// TwinCAT 3 PLC project PLC1
// ProgramVersion: 3.1.4022.2
// libraries:
//   Tc2_DALI, * (Beckhoff Automation GmbH)
//   Tc2_EnOcean, * (Beckhoff Automation GmbH)
//   Tc2_IoFunctions, * (Beckhoff Automation GmbH)
//   Tc2_ModbusRTU, * (Beckhoff Automation GmbH)
//   Tc2_ModbusSrv, * (Beckhoff Automation GmbH)
//   Tc2_Standard, * (Beckhoff Automation GmbH)
//   Tc2_System, * (Beckhoff Automation GmbH)
//   Tc3_Module, * (Beckhoff Automation GmbH)
//   Tc3_PLCopen_OpcUa, * (Beckhoff Automation GmbH)
//   VisuSymbols,3.5.10.0,System
// project tree:
//   / DaliComm.TcTTO, GlobalTextList.TcGTLO, IoConversionTask.TcTTO, ModbusComm.TcTTO, PlcTask.TcTTO, Visualization Manager.TcVMO (not stored)
//   DUTs/ ATV212.TcDUT, ATV212Control.TcDUT, ATV212RegAddress.TcDUT, EL3433Index.TcDUT, EL3433Measurement.TcDUT, ErrorCode.TcDUT, Fan.TcDUT, FireIgnitor.TcDUT, GrundfosMagna3.TcDUT, GrundfosRegAddress.TcDUT, stEL3433_In.TcDUT, SupplyCondition.TcDUT
//   GVLs/ ConstList.TcGVL, GVL.TcGVL, HWVar.TcGVL, Scale.TcGVL
//   POUs/BurningProcess/ BurningProcess.TcPOU, FB_OnOffTimer.TcPOU (not stored), FeederSpeedControl.TcPOU
//   POUs/CommunicationPrograms/ BackgroundComm.TcPOU, DaliCommunication.TcPOU, EL3433SyncData.TcPOU, IOConversion.TcPOU
//   POUs/EnergyFlow/ CoolingFan.TcPOU, WaterFlowControl.TcPOU
//   POUs/Lights/ EnOcean_Dali.TcPOU
//   POUs/ MAIN.TcPOU, ModbusCommunication.TcPOU
// real-time tasks:
//   TASK PlcTask: cycle T#5ms, priority 20, ADS port 350
//   TASK ModbusComm: cycle T#5ms, priority 21, ADS port 351
//   TASK IoConversionTask: cycle T#1ms, priority 10, ADS port 352
//   TASK DaliComm: cycle T#1ms, priority 15, ADS port 353
// I/O:
//   DEVICE Device 1 (EtherCAT), AmsNetId 5.42.255.222.2.1
//     Term 1 (EK1200) [EK1200-5000 EtherCAT Power supply (2A E-Bus)]
//       Term 2 (EL1008) [EL1008 8Ch. Dig. Input 24V, 3ms]
//       Term 3 (EL6021) [EL6021 Interface (RS422/485)]
//       Term 4 (EK1122) [EK1122 2 port EtherCAT junction]
//         Term 5 (EK1914) [EK1914, 2 Ch. Safety Input/Output 24V,  TwinSAFE]
//           modules: Module 1 (FSOE), Module 2 (DIO)
//           Term 6 (EL2809) [EL2809 16Ch. Dig. Output 24V, 0.5A]
//           Term 7 (EL3214) [EL3214 4Ch. Ana. Input PT100 (RTD)]
//           Term 24 (EL3204) [EL3204 4Ch. Ana. Input PT100 (RTD)]
//           Term 16 (EL9011) [EL9011 End Terminal]
//         Term 8 (EK1100) [EK1100 EtherCAT Coupler (2A E-Bus)]
//           Term 9 (EL6021) [EL6021 Interface (RS422/485)]
//           Term 10 (EL2008) [EL2008 8Ch. Dig. Output 24V, 0.5A]
//           Term 11 (EL4022) [EL4022 2Ch. Ana. Output 4-20mA, 12bit]
//           Box 12 (BK1250)
//       Term 13 (EL3433) [EL3433 3Ch. Power Measuring]
//       Term 14 (EL3433) [EL3433 3Ch. Power Measuring]
//       Box 15 (BK1250)
// variable links:
//   PLC1/PLC1 Instance <-> Device 1 (EtherCAT)/Term 1 (EK1200)/Box 15 (BK1250)
//     DaliComm Inputs/HWVar.stKL6811_in/nData <-> Term 8 (KL6811)/Channel 1/Data In
//     DaliComm Inputs/HWVar.stKL6811_in/nStatus <-> Term 8 (KL6811)/Channel 1/State
//     DaliComm Outputs/HWVar.stKL6811_out/nCtrl <-> Term 8 (KL6811)/Channel 1/Ctrl
//     DaliComm Outputs/HWVar.stKL6811_out/nData <-> Term 8 (KL6811)/Channel 1/Data Out
//     PlcTask Inputs/HWVar.st6581_in @bit 8 <-> Term 7 (KL6581)/Channel 1/Input CNODE
//     PlcTask Inputs/HWVar.st6581_in @bit {24..48 step 8} <-> Term 7 (KL6581)/Channel 1/Input DB{0..3}  (4 links)
//     PlcTask Inputs/HWVar.st6581_in @bit {56..80 step 8} <-> Term 7 (KL6581)/Channel 1/Input ID{0..3}  (4 links)
//     PlcTask Inputs/HWVar.st6581_in @bit 16 <-> Term 7 (KL6581)/Channel 1/Input ORG
//     PlcTask Inputs/HWVar.st6581_in @bit 88 <-> Term 7 (KL6581)/Channel 1/Input STATUS
//     PlcTask Inputs/HWVar.st6581_in <-> Term 7 (KL6581)/Channel 1/Status
//     PlcTask Outputs/HWVar.st6581_out <-> Term 7 (KL6581)/Channel 1/Control
//     PlcTask Outputs/HWVar.st6581_out @bit 8 <-> Term 7 (KL6581)/Channel 1/Output CNODE
//     PlcTask Outputs/HWVar.st6581_out @bit {24..48 step 8} <-> Term 7 (KL6581)/Channel 1/Output DB{0..3}  (4 links)
//     PlcTask Outputs/HWVar.st6581_out @bit {56..80 step 8} <-> Term 7 (KL6581)/Channel 1/Output ID{0..3}  (4 links)
//     PlcTask Outputs/HWVar.st6581_out @bit 16 <-> Term 7 (KL6581)/Channel 1/Output ORG
//     PlcTask Outputs/HWVar.st6581_out @bit 88 <-> Term 7 (KL6581)/Channel 1/Output STATUS
//   PLC1/PLC1 Instance <-> Device 1 (EtherCAT)/Term 1 (EK1200)/Term 13 (EL3433)
//     IoConversionTask Inputs/HWVar.EL3433_Grid[1]/dCurrent <-> PM Inputs Channel 1/Current
//     IoConversionTask Inputs/HWVar.EL3433_Grid[2]/dCurrent <-> PM Inputs Channel 2/Current
//     IoConversionTask Inputs/HWVar.EL3433_Grid[3]/dCurrent <-> PM Inputs Channel 3/Current
//     IoConversionTask Inputs/HWVar.EL3433_Grid[1]/dIndex <-> PM Inputs Channel 1/Index
//     IoConversionTask Inputs/HWVar.EL3433_Grid[2]/dIndex <-> PM Inputs Channel 2/Index
//     IoConversionTask Inputs/HWVar.EL3433_Grid[3]/dIndex <-> PM Inputs Channel 3/Index
//     IoConversionTask Inputs/HWVar.EL3433_Grid[1]/dPower <-> PM Inputs Channel 1/Active power
//     IoConversionTask Inputs/HWVar.EL3433_Grid[2]/dPower <-> PM Inputs Channel 2/Active power
//     IoConversionTask Inputs/HWVar.EL3433_Grid[3]/dPower <-> PM Inputs Channel 3/Active power
//     IoConversionTask Inputs/HWVar.EL3433_Grid[1]/dVariant <-> PM Inputs Channel 1/Variant value
//     IoConversionTask Inputs/HWVar.EL3433_Grid[2]/dVariant <-> PM Inputs Channel 2/Variant value
//     IoConversionTask Inputs/HWVar.EL3433_Grid[3]/dVariant <-> PM Inputs Channel 3/Variant value
//     IoConversionTask Inputs/HWVar.EL3433_Grid[1]/dVoltage <-> PM Inputs Channel 1/Voltage
//     IoConversionTask Inputs/HWVar.EL3433_Grid[2]/dVoltage <-> PM Inputs Channel 2/Voltage
//     IoConversionTask Inputs/HWVar.EL3433_Grid[3]/dVoltage <-> PM Inputs Channel 3/Voltage
//     IoConversionTask Outputs/HWVar.EL3433_GridIndex[1] <-> PM Outputs Channel 1/Index
//     IoConversionTask Outputs/HWVar.EL3433_GridIndex[2] <-> PM Outputs Channel 2/Index
//     IoConversionTask Outputs/HWVar.EL3433_GridIndex[3] <-> PM Outputs Channel 3/Index
//   PLC1/PLC1 Instance <-> Device 1 (EtherCAT)/Term 1 (EK1200)/Term 14 (EL3433)
//     IoConversionTask Inputs/HWVar.EL3433_Solar/dCurrent <-> PM Inputs Channel 1/Current
//     IoConversionTask Inputs/HWVar.EL3433_Solar/dIndex <-> PM Inputs Channel 1/Index
//     IoConversionTask Inputs/HWVar.EL3433_Solar/dPower <-> PM Inputs Channel 1/Active power
//     IoConversionTask Inputs/HWVar.EL3433_Solar/dVariant <-> PM Inputs Channel 1/Variant value
//     IoConversionTask Inputs/HWVar.EL3433_Solar/dVoltage <-> PM Inputs Channel 1/Voltage
//     IoConversionTask Outputs/HWVar.EL3433_SolarIndex <-> PM Outputs Channel 1/Index
//   PLC1/PLC1 Instance <-> Device 1 (EtherCAT)/Term 1 (EK1200)/Term 3 (EL6021)
//     PlcTask Inputs/HWVar.ModbusMaster1.InData @bit {16..184 step 8} <-> COM TxPDO-Map Inputs/Data In {0..21}  (22 links)
//     PlcTask Inputs/HWVar.ModbusMaster1.InData <-> COM TxPDO-Map Inputs/Status
//     PlcTask Outputs/HWVar.ModbusMaster1.OutData <-> COM RxPDO-Map Outputs/Ctrl
//     PlcTask Outputs/HWVar.ModbusMaster1.OutData @bit {16..184 step 8} <-> COM RxPDO-Map Outputs/Data Out {0..21}  (22 links)
//   PLC1/PLC1 Instance <-> Device 1 (EtherCAT)/Term 1 (EK1200)/Term 4 (EK1122)/Term 5 (EK1914)/Term 24 (EL3204)
//     IoConversionTask Inputs/HWVar.iAI2_VK[{1..4}] <-> RTD Inputs Channel {1..4}/Value  (4 links)
//   PLC1/PLC1 Instance <-> Device 1 (EtherCAT)/Term 1 (EK1200)/Term 4 (EK1122)/Term 5 (EK1914)/Term 6 (EL2809)
//     PlcTask Outputs/GVL.bFanPower <-> Channel 12/Output
//     PlcTask Outputs/GVL.bHV[{2..11}] <-> Channel {2..11}/Output  (10 links)
//     PlcTask Outputs/GVL.bHV[1] <-> Channel 1/GVL.bHV[1]
//   PLC1/PLC1 Instance <-> Device 1 (EtherCAT)/Term 1 (EK1200)/Term 4 (EK1122)/Term 5 (EK1914)/Term 7 (EL3214)
//     IoConversionTask Inputs/HWVar.iAI1_VK[{1..4}] <-> RTD Inputs Channel {1..4}/HWVar.iAI1_VK[{1..4}]  (4 links)
//   PLC1/PLC1 Instance <-> Device 1 (EtherCAT)/Term 1 (EK1200)/Term 4 (EK1122)/Term 8 (EK1100)/Box 12 (BK1250)
//     IoConversionTask Inputs/HWVar.iAI1_JK[{1..4}] <-> Term 5 (KL3204)/Channel {1..4}/Data In  (4 links)
//     IoConversionTask Inputs/HWVar.iKL3064[{1..4}] <-> Term 17 (KL3064)/Channel {1..4}/HWVar.iKL3064[{1..4}]  (4 links)
//     IoConversionTask Inputs/HWVar.stKL2761_in/iDataIn <-> Term 15 (KL2761)/Channel 1/Data In
//     IoConversionTask Inputs/HWVar.stKL2761_in/iState <-> Term 15 (KL2761)/Channel 1/State
//     IoConversionTask Inputs/HWVar.stKL3208_in/iDataIn <-> Term 3 (KL3208-0010-4)/Channel 1/Data In
//     IoConversionTask Inputs/HWVar.stKL3208_in/iState <-> Term 3 (KL3208-0010-4)/Channel 1/State
//     IoConversionTask Outputs/HWVar.stKL2761_out/iCtrl <-> Term 15 (KL2761)/Channel 1/Ctrl
//     IoConversionTask Outputs/HWVar.stKL2761_out/iDataOut <-> Term 15 (KL2761)/Channel 1/Data Out
//     ModbusComm Outputs/HWVar.stKL3204_out/iCtrl <-> Term 5 (KL3204)/Channel 4/Ctrl
//     ModbusComm Outputs/HWVar.stKL3204_out/iDataOut <-> Term 5 (KL3204)/Channel 4/Data Out
//     PlcTask Outputs/HWVar.stKL3208_out/iCtrl <-> Term 3 (KL3208-0010-4)/Channel 1/Ctrl
//     PlcTask Outputs/HWVar.stKL3208_out/iDataOut <-> Term 3 (KL3208-0010-4)/Channel 1/Data Out
//   PLC1/PLC1 Instance <-> Device 1 (EtherCAT)/Term 1 (EK1200)/Term 4 (EK1122)/Term 8 (EK1100)/Term 10 (EL2008)
//     PlcTask Outputs/GVL.stFI1/bBlower <-> Channel 5/Output
//     PlcTask Outputs/GVL.stFI1/bHeating <-> Channel 3/Output
//   PLC1/PLC1 Instance <-> Device 1 (EtherCAT)/Term 1 (EK1200)/Term 4 (EK1122)/Term 8 (EK1100)/Term 9 (EL6021)
//     PlcTask Inputs/HWVar.ModbusMaster.InData/D <-> COM TxPDO-Map Inputs/Data In 0
//     PlcTask Inputs/HWVar.ModbusMaster.InData/D @bit {8..168 step 8} <-> COM TxPDO-Map Inputs/Data In {1..21}  (21 links)
//     PlcTask Inputs/HWVar.ModbusMaster.InData/Status <-> COM TxPDO-Map Inputs/Status
//     PlcTask Outputs/HWVar.ModbusMaster.OutData/Ctrl <-> COM RxPDO-Map Outputs/Ctrl
//     PlcTask Outputs/HWVar.ModbusMaster.OutData/D <-> COM RxPDO-Map Outputs/Data Out 0
//     PlcTask Outputs/HWVar.ModbusMaster.OutData/D @bit {8..168 step 8} <-> COM RxPDO-Map Outputs/Data Out {1..21}  (21 links)

CONFIGURATION PLC1
    RESOURCE PLC ON TwinCAT3
        TASK DaliComm(INTERVAL := T#1ms, PRIORITY := 15);
        TASK IoConversionTask(INTERVAL := T#1ms, PRIORITY := 10);
        TASK ModbusComm(INTERVAL := T#5ms, PRIORITY := 21);
        TASK PlcTask(INTERVAL := T#5ms, PRIORITY := 20);
        PROGRAM DaliCommunication WITH DaliComm : DaliCommunication;
        PROGRAM IOConversion WITH IoConversionTask : IOConversion;
        PROGRAM BackgroundComm WITH ModbusComm : BackgroundComm;
        PROGRAM MAIN WITH PlcTask : MAIN;
    END_RESOURCE
END_CONFIGURATION

// ---- DUTs/ATV212.TcDUT
{attribute 'pack_mode' := '1'}
TYPE ATV212 :
STRUCT
	fMotorSpeed				: REAL;
	fOutputFrequency		: REAL;
	fOutputCurrent			: REAL;
	fOutputVoltage			: REAL;
END_STRUCT
END_TYPE

// ---- DUTs/ATV212Control.TcDUT
{attribute 'pack_mode' := '1'}
TYPE ATV212Control :
STRUCT
	bStart		: BOOL;
	bForward	: BOOL;
	fFrequency	: REAL;
	bManual		: BOOL;
	tTimeOn		: TIME;
	tTimeOff	: TIME;
END_STRUCT
END_TYPE

// ---- DUTs/ATV212RegAddress.TcDUT
{attribute 'qualified_only'}
TYPE ATV212RegAddress :
(
               listStart                        := 16#1874,
               MotorSpeed                       := 16#1875,
               Frequency                       	:= 16#1876,
               Current                        	:= 16#1877,
               Voltage                        	:= 16#1878,
               
               (*
               OutputFrequencyAtLastTrip		:= 16#FE00, // Hz Value before trip
               FrequencyReferenceBeforeRamp     := 16#FE02, // Hz Value before trip (before PI and speed ramp)
               FrequencyReferenceAfterRamp      := 16#FE15, // Hz Value before trip (after PI AND speed ramp)
               EstimatedSpeed                   := 16#FE16, // Hz Value before trip
               PIDFeedbackValue                 := 16#FE22, // Hz Value before trip
               
               
               
               Torque                           := 16#FE18,
               TorqueCurrent                    := 16#FE20,  //Value before trip
               ExcitingCurrent                  := 16#FE21,  //Value before trip*)
			   listEnd                          := 16#1879
) WORD := listStart;
END_TYPE

// ---- DUTs/EL3433Index.TcDUT
{attribute 'qualified_only'}
TYPE EL3433Index :
(	
	listStart := 3,
	ApparentPower :=3,
	Q,
	Energy,
	PF,
	Frequency,
	EnergyNegative,
	PhaseAngle,
	P1,
	S1,
	Q1,
	EnergyPositive,
	EnergyPositiveSaved,
	EnergySaved,
	EnergyNegativeSaved,
	FrequencyAvgRes,
	FrequencyHiRes,
	HeldFrequency,
	HeldFrequencyAvgRes,
	HeldFrequencyHiRes,
	listEnd := HeldFrequencyHiRes
);
END_TYPE

// ---- DUTs/EL3433Measurement.TcDUT
{attribute 'pack_mode' := '1'}
TYPE EL3433Measurement :
STRUCT
	fCurrent		: REAL;
	fVoltage		: REAL;
	fP		: REAL;
	fS		: REAL;
	fQ		: REAL;
	fEnergy		: REAL;
	fPF		: REAL;
	fFrequency		: REAL;
	fEnergyNegative		: REAL;
	fPhaseAngle		: REAL;
	fP1		: REAL;
	fS1		: REAL;
	fQ1		: REAL;
	fEnergyPositive		: REAL;
	fEnergyPositiveSaved		: REAL;
	fEnergySaved		: REAL;
	fEnergyNegativeSaved		: REAL;
	fFrequencyAvgRes		: REAL;
	fFrequencyHiRes		: REAL;
	fHeldFrequency		: REAL;
	fHeldFrequencyAvgRes		: REAL;
	fHeldFrequencyHiRes		: REAL;
END_STRUCT
END_TYPE

// ---- DUTs/ErrorCode.TcDUT
{attribute 'qualified_only'}
TYPE ErrorCode :
(
	SUCCESS := 0,
	
	// Preparation Error 
	PREPARATION_DONE := 1000,
	PREPARATION_WATER_HIGH_TEMP,
	PREPARATION_FLAME,
	PREPARATION_PUMP_NOT_CONNECTED,
	
	// Ignition Error
	IGNITION_DONE := 2000,
	IGNITION_FLAME,
	
	// Burning Error
	BURNING_DONE := 3000,
	BURNING_EMERGENCY_TEMPERATURE,
	
	// Stop Error
	STOP_ERROR	:= 4000
) UINT;
END_TYPE

// ---- DUTs/Fan.TcDUT
{attribute 'pack_mode' := '1'}
TYPE Fan :
STRUCT
	nSpeed 	: INT; // control primary fan speed 0-100%
	nTemp	: INT; // prim fan's terminal temp in Celcius
	fFE		: REAL;
END_STRUCT
END_TYPE

// ---- DUTs/FireIgnitor.TcDUT
{attribute 'pack_mode' := '1'}
TYPE FireIgnitor :
STRUCT
	bHeating				: BOOL;
	bBlower					: BOOL;
END_STRUCT
END_TYPE

// ---- DUTs/GrundfosMagna3.TcDUT
{attribute 'pack_mode' := '1'}
TYPE GrundfosMagna3 :
STRUCT
	fHead                       : REAL; 
	fVolumeFlow                 : REAL;
	fRelativePerformance        : REAL;
	fSpeed                      : REAL;
	fFrequency                  : REAL;
	fDigitalInput               : REAL;
	fDigitalOutput              : REAL;
	fActualSetpoint             : REAL;
	fMotorCurrent               : REAL;
	fDCLinkVoltage              : REAL;
	fMotorVoltage			    : REAL;
	fPower                      : REAL;
	fRemoteFlow                 : REAL;
	fInletPressure              : REAL;
    fRemotePressure             : REAL;
	fLevel                      : REAL;
	fPowerElectronicTemp        : REAL;
	fMotorTemp                  : REAL;
	fRemoteTemp                 : REAL;
	fElectronicTemp             : REAL;
	fPumpLiquidTemp             : REAL;
	fBearingTempDE			    : REAL;
	fBearingTempNDE             : REAL;
    fAuxSensorInput             : REAL;
    fSpecificEnergyConsumption  : REAL;
    fOperationTime              : REAL;         
    fTotalPoweredTime           : REAL;
    fTorque                     : REAL;
    fEnergy                     : REAL;
    fNumberOfStarts             : REAL;
    fReserved1                  : REAL;
    fRemoteTemp2                : REAL;
    fUserSetpoint               : REAL;
    fDiffPressure               : REAL;
    fOutletPressure             : REAL;
    fRemotePressure2            : REAL;
    fLoadPercent                : REAL;
    fPumpUnixRtc                : REAL;
    fMaxFlowLimit               : REAL;
    fRemoteDiffTemp             : REAL;
    fInletDiffPressure          : REAL;
    fOutletDiffPressure         : REAL;
    fRemoteDiffPressure         : REAL;
    fStorageTankLevel           : REAL;
    fAmbientTemp                : REAL;
    fHeatEnergyLifetime         : REAL;
    fHeatPower                  : REAL;
    fHeatDiffTemp               : REAL;
    fVolume                     : REAL;
    fHeatEnergyCounter2         : REAL;
    fVolume2                    : REAL;
END_STRUCT
END_TYPE

// ---- DUTs/GrundfosRegAddress.TcDUT
{attribute 'qualified_only'}
TYPE GrundfosRegAddress :
(
	listStart				   := 299,
	Head                       := 300, 
	VolumeFlow                 ,
	RelativePerformance        ,
	Speed                      ,
	Frequency                  ,
	DigitalInput               ,
	DigitalOutput              ,
	ActualSetpoint             ,
	MotorCurrent               ,
	DCLinkVoltage              ,
	MotorVoltage			   ,
	Power                      ,
	RemoteFlow                 := 313,
	InletPressure              ,
    RemotePressure             ,
	Level                      ,
	PowerElectronicTemp        ,
	MotorTemp                  ,
	RemoteTemp                 ,
	ElectronicTemp             ,
	PumpLiquidTemp             ,
	BearingTempDE			   ,
	BearingTempNDE             ,
    AuxSensorInput             ,
    SpecificEnergyConsumption  ,
    OperationTime              ,         
    TotalPoweredTime           := 328,
    Torque                     := 330,
    Energy                     ,
    NumberOfStarts             := 333,
    Reserved1                  := 335,
    RemoteTemp2                ,
    UserSetpoint               ,
    DiffPressure               ,
    OutletPressure             ,
    RemotePressure2            ,
    LoadPercent                ,
    PumpUnixRtc                ,
    MaxFlowLimit               := 344,
    RemoteDiffTemp             ,
    InletDiffPressure          ,
    OutletDiffPressure         ,
    RemoteDiffPressure         ,
    StorageTankLevel           ,
    AmbientTemp                ,
    HeatEnergyLifetime         ,
    HeatPower                  := 353,
    HeatDiffTemp               := 355,
    Volume                     ,
    HeatEnergyCounter2         := 358,
    Volume2                    := 360,
	listEnd					   := 361
) WORD := listStart;
END_TYPE

// ---- DUTs/stEL3433_In.TcDUT
{attribute 'pack_mode' := '1'}
TYPE stEL3433_In :
STRUCT
	dCurrent 	:	DINT;
	dVoltage 	:	DINT;
	dPower		:	DINT;
	dIndex 		:	USINT;
	dVariant	:	DINT;
END_STRUCT
END_TYPE

// ---- DUTs/SupplyCondition.TcDUT
{attribute 'pack_mode' := '1'}
TYPE SupplyCondition :
STRUCT
	fNeutralConductorCurrent				:REAL;
	fEnergySum				:REAL;
	fFrequency				:REAL;
	fNegativeEnergySum				:REAL;
	fPSum				:REAL;
	fSSum				:REAL;
	fQSum				:REAL;
	fFundamentalP				:REAL;
	fFundamentalS				:REAL;
	fFundamentalQ				:REAL;
	fEnergyPositive				:REAL;
	fEnergyPositiveSaved				:REAL;
	fEnergyNegative				:REAL;
	fEnergyNegativeSaved				:REAL;
	fFrequencyAvgRes				:REAL;
	fFrequencyHiRes				:REAL;
	fHeldFrequency				:REAL;
	fHeldFrequencyAvgRes				:REAL;
	fHeldFrequencyHiRes				:REAL;
	fADCTemperature				:REAL;

END_STRUCT
END_TYPE

// ---- GVLs/ConstList.TcGVL
VAR_GLOBAL
	aEL3433IndicesScale	: ARRAY[EL3433Index.listStart..EL3433Index.listEnd]	OF REAL := [
		0.01,
		0.01,
		0.001,
		0.001,
		0.1,
		0.001,
		0.01,
		0.01,
		0.01,
		0.01,
		0.001,
		0.001,
		0.001,
		0.001,
		0.01,
		0.001,
		0.1,
		0.01,
		0.001
	];
	aEL3433Indices	: ARRAY[EL3433Index.listStart..EL3433Index.listEnd]	OF  USINT := [
		0,
		1,
		2,
		3,
		4,
		5,
		6,
		20,
		21,
		22,
		30,
		31,
		32,
		35,
		44,
		45,
		46,
		47,
		48
	];
	WaterTempMax	: INT 	:= 85; // Maximum water temperature
	WaterTempMin	: INT	:= 60; // Minimum water temperature
	WaterTempDes	: INT	:= 75; // Desired water temperature
	WaterTempWar	: INT	:= 90; // Warning water temperature
END_VAR

// ---- GVLs/GVL.TcGVL
{attribute 'qualified_only'}
VAR_GLOBAL
	{attribute 'OPC.UA.DA' := '1'}
	fTE         : ARRAY [1..22] OF REAL;
	{attribute 'OPC.UA.DA' := '1'}
    bHV AT %Q*  : ARRAY [1..11] OF BOOL;
	{attribute 'OPC.UA.DA' := '1'}
	bFanPower AT %Q* : BOOL;  // Lauhdutin fan power
	{attribute 'OPC.UA.DA' := '1'}
    bP1	: BOOL := TRUE;
	{attribute 'OPC.UA.DA' := '1'}
    bP2	: BOOL := TRUE;
	{attribute 'OPC.UA.DA' := '1'}
    bP3	: BOOL := TRUE;
	{attribute 'OPC.UA.DA' := '1'}
	stP1		: GrundfosMagna3;
	{attribute 'OPC.UA.DA' := '1'}
	stP2		: GrundfosMagna3;
	{attribute 'OPC.UA.DA' := '1'}
	stP3		: GrundfosMagna3;
	{attribute 'OPC.UA.DA' := '1'}
	stFeeder	: ATV212;
	{attribute 'OPC.UA.DA' := '1'}
	stFeederControl : ATV212Control;
	{attribute 'OPC.UA.DA' := '1'}
	bLoadTank1	: BOOL := TRUE;
	{attribute 'OPC.UA.DA' := '1'}
	bLoadTank2	: BOOL := TRUE;
	{attribute 'OPC.UA.DA' := '1'}
	bLoadTank3	: BOOL := TRUE;
	{attribute 'OPC.UA.DA' := '1'}
	stMain	: ARRAY [1..3] OF EL3433Measurement; 
	{attribute 'OPC.UA.DA' := '1'}
	stSolarL1	: EL3433Measurement;
	{attribute 'OPC.UA.DA' := '1'}
	nError	: UINT; 
	{attribute 'OPC.UA.DA' := '1'}
	nFlame		: REAL;
	{attribute 'OPC.UA.DA' := '1'}
	stPrimaryFan	: FAN;
	{attribute 'OPC.UA.DA' := '1'}
	stSecondaryFan	: FAN;
	{attribute 'OPC.UA.DA' := '1'}
	bValveManual	: BOOL; // load tank manually or automatically based on water temps
	{attribute 'OPC.UA.DA' := '1'}
	bBurningStart : BOOL;
	{attribute 'OPC.UA.DA' := '1'}
	stFI1	AT %Q* : FireIgnitor;
	{attribute 'OPC.UA.DA' := '1'}
	fO2	:	REAL;
END_VAR

// ---- GVLs/HWVar.TcGVL
{attribute 'qualified_only'}
VAR_GLOBAL
	stKL3204_in     AT %I*  : ST_KL320xInData ;
	stKL3204_out    AT %Q*  : ST_KL320xOutData ;
    iAI1_VK         AT %I*  : ARRAY [1..4] OF INT;
    iAI2_VK         AT %I*  : ARRAY [1..4] OF INT;
    iAI1_JK         AT %I*  : ARRAY [1..4] OF INT;
    ModbusMaster            : ModbusRtuMaster_KL6x22B;
	ModbusMaster1           : ModbusRtuMaster_KL6x22B;
	EL3433_Grid		AT %I*	: ARRAY[1..3] OF stEL3433_In;
	EL3433_GridIndex AT %Q*	: ARRAY[1..3] OF USINT;
	EL3433_SolarIndex AT %Q*: USINT;
	EL3433_Solar 	AT %I*	: stEL3433_In;
	// Enocean valiables	
	st6581_in		AT %I*	: KL6581_Input;
	st6581_out		AT %Q*	: KL6581_Output;
	stKL6581				: STR_KL6581;
	// Dali variables
	//	stKL6811_in     AT %I*	: ST_DALIV2InData;
	stKL6811_in     AT %I*	: ST_KL6811InData;
	//    stKL6811_out    AT %Q*	: ST_DALIV2OutData;
    stKL6811_out    AT %Q*	: ST_KL6811OutData;
	stKL6811_CommandBuffer  : ST_DALIV2CommandBuffer;
	//	DaliMaster				: FB_DALIV2Communication;
	DaliMaster				: FB_KL6811Communication;
	bDaliReset : BOOL;
	
	stKL2761_in		AT %I* 	: ST_KL27x1InData; // Primary fan input
	stKL2761_out	AT %Q* 	: ST_KL27x1OutData; //Primary fan output
	
	stKL3208_in		AT %I*	: ST_KL3208InData;  //8-channel input terminal PT1000, Ni1000 (RTD); NTC sensors, potentiometers
	stKL3208_out	AT %Q*	: ST_KL3208OutData;
	
	// analog DC input HW 
	iKL3064			AT %I*	: ARRAY [1..4] OF INT;
	
 
END_VAR

// ---- GVLs/Scale.TcGVL
{attribute 'qualified_only'}
VAR_GLOBAL
	fGrundfosScale	: ARRAY [300..350] OF REAL := [
		0.001,		//Head                        
		0.1,		//VolumeFlow                 
		0.01,		//RelativePerformance        
		1.0,		//Speed                      
		0.1,		//Frequency                  
		1.0,		//DigitalInput               
		1.0,		//DigitalOutput              
		0.01,		//ActualSetpoint             
		0.1,		//MotorCurrent               
		0.1,		//DCLinkVoltage              
		0.1,		//MotorVoltage			    
		1.0,		//Power                      
		0.1,		//RemoteFlow                 
		0.001,		//InletPressure              
		0.001,		//RemotePressure             
		0.01,		//Level                      
		0.01,		//PowerElectronicTemp        
		0.01,		//MotorTemp                  
		0.01,		//RemoteTemp                 
		0.01,		//ElectronicTemp             
		0.01,		//PumpLiquidTemp             
		0.01,		//BearingTempDE			    
		0.01,		//BearingTempNDE             
		0.01,		//AuxSensorInput             
		1.0,		//SpecificEnergyConsumption  
		1.0,		//OperationTime                       
		1.0,		//TotalPoweredTime           
		0.1,		//Torque                     
		1.0,		//Energy                     
		1.0,		//NumberOfStarts             
		1.0,		//Reserved1                  
		0.01,		//RemoteTemp2                
		0.01,		//UserSetpoint               
		0.001,		//DiffPressure               
		0.001,		//OutletPressure             
		0.001,		//RemotePressure2            
		0.01,		//LoadPercent                
		1.0,		//PumpUnixRtc                
		0.1,		//MaxFlowLimit               
		0.01,		//RemoteDiffTemp             
		0.001,		//InletDiffPressure          
		0.001,		//OutletDiffPressure         
		0.001,		//RemoteDiffPressure         
		0.01,		//StorageTankLevel           
		0.01,		//AmbientTemp                
		1.0,		//HeatEnergyLifetime         
		1.0,		//HeatPower                  
		0.01,		//HeatDiffTemp               
		0.01,		//Volume                     
		1.0,		//HeatEnergyCounter2         
		0.01		//Volume2                    
	];
	fATV212Scale     : ARRAY [ATV212RegAddress.listStart +1 ..ATV212RegAddress.listEnd -1 ] OF REAL := [
    	1,          //Motor Speed                        
    	0.01,       //Output frequency                
    	0.01,       //Output current
    	0.01        //Output votlage
    ];
END_VAR

// ---- POUs/CommunicationPrograms/DaliCommunication.TcPOU
PROGRAM DaliCommunication
VAR
	arrBufferDemandMeter: ARRAY [0..2] OF BYTE;
	arrBufferMaximumDemandMeter: ARRAY [0..2] OF BYTE;
	arrBufferOverflowCounter: ARRAY [0..2] OF UINT;
	bLineIsBusy: BOOL;
	bLineIsInitialized: BOOL;
END_VAR

HWVar.DaliMaster(
	bResetMaximumDemandCounter:= HWVar.bDaliReset, 
	bResetOverflowCounter:= HWVar.bDaliReset, 
	arrBufferDemandMeter=> arrBufferDemandMeter, 
	arrBufferMaximumDemandMeter=> arrBufferMaximumDemandMeter, 
	arrBufferOverflowCounter=> arrBufferOverflowCounter, 
	bLineIsBusy=> bLineIsBusy, 
	bLineIsInitialized=> bLineIsInitialized, 
	stDALIInData:= HWVar.stKL6811_in, 
	stDALIOutData:= HWVar.stKL6811_out, 
	stCommandBuffer:= HWVar.stKL6811_CommandBuffer);

END_PROGRAM

// ---- POUs/CommunicationPrograms/IOConversion.TcPOU
PROGRAM IOConversion
VAR
	i: INT;
	EL3433DataMain 	: ARRAY[1..3] OF EL3433SyncData;
	EL3433DataSolar	: EL3433SyncData;
	nFlowVoltage, nO2Voltage: REAL;
END_VAR

GVL.fTE[1] := HWVar.iAI1_VK[4]/10.0; // from solar to kattila temp
GVL.fTE[18] := HWVar.iAI1_JK[1]/10.0; // from kattila to solar temp

GVL.fTE[5] := HWVar.iAI1_JK[2]/10.0; // kattila out temp
GVL.fTE[6] := HWVar.iAI1_VK[3]/10.0; // tank1 in temp
GVL.fTE[7] := HWVar.iAI1_VK[2]/10.0; // tank2 in temp
GVL.fTE[8] := HWVar.iAI1_VK[1]/10.0; // tank8 in temp

GVL.fTE[15] := HWVar.iAI2_VK[1]/10.0; // lauhdutin in temp 
GVL.fTE[16] := HWVar.iAI2_VK[3]/10.0; // lauhdutin out temp

GVL.fTE[19] := HWVar.iAI1_JK[3]/10.0; // exhaust temp
GVL.fTE[17] := HWVar.iAI1_JK[4]/10.0; // kattila room temp

GVL.fTE[20] := HWVar.stKL3208_in.iDataIn/1000.0; // kattila room temp

nFlowVoltage := INT_TO_REAL(HWVar.iKL3064[1])*0.0003 + 0.0008; // 12 bits, output 0.525-2.6V, range 0-1L/s
GVL.stPrimaryFan.fFE := (46.606*EXPT(nFlowVoltage,3) - 181.24*EXPT(nFlowVoltage,2) + 258.22*nFlowVoltage -93.735) * 1000 / 3600 ;

GVL.fO2 := INT_TO_REAL(HWVar.iKL3064[4])*10/32767*21/5; // 12 bits, output 0.525-2.6V, range 0-1L/s


GVL.stPrimaryFan.nTemp := HWVar.stKL2761_in.iDataIn; //read prim fan terminal temp
HWVar.stKL2761_out.iDataOut := GVL.stPrimaryFan.nSpeed*32767/100; //control prim fan speed

FOR i:= 1 TO 3 DO
	GVL.stMain[i].fCurrent := TO_REAL(HWVar.EL3433_Grid[i].dCurrent)*0.000001;
	GVL.stMain[i].fVoltage := TO_REAL(HWVar.EL3433_Grid[i].dVoltage)*0.0001;
	GVL.stMain[i].fP := TO_REAL(HWVar.EL3433_Grid[i].dPower)*0.01;
	EL3433DataMain[i](
		pstEL3433Data := ADR(GVL.stMain[i]),
		pstEL3433IO := ADR(HWVar.EL3433_Grid[i]),
		pstEL3433OutputIndex := ADR(HWVar.EL3433_GridIndex[i])
	);
END_FOR
GVL.stSolarL1.fCurrent := TO_REAL(HWVar.EL3433_Solar.dCurrent)*0.000001;
GVL.stSolarL1.fVoltage := TO_REAL(HWVar.EL3433_Solar.dVoltage)*0.0001;
GVL.stSolarL1.fP := TO_REAL(HWVar.EL3433_Solar.dPower)*0.01;
	EL3433DataSolar(
		pstEL3433Data := ADR(GVL.stSolarL1),
		pstEL3433IO := ADR(HWVar.EL3433_Solar),
		pstEL3433OutputIndex := ADR(HWVar.EL3433_SolarIndex)
	);
//EL3433DAQ(ADR(GVL.stMain[1]],ADR(HWVar.EL3433_Grid[1]),ADR(HWVar.EL3433_GridIndex[1]));

END_PROGRAM

// ---- POUs/CommunicationPrograms/EL3433SyncData.TcPOU
FUNCTION_BLOCK EL3433SyncData
VAR_INPUT
	pstEL3433Data	: POINTER TO EL3433Measurement;
	pstEL3433IO		: POINTER TO stEL3433_In;
	pstEL3433OutputIndex	: POINTER TO USINT;
END_VAR

VAR
	pTempReal	: POINTER TO REAL;
	nArrayIndex	: DWORD := TO_DWORD(EL3433Index.listStart);
END_VAR

VAR_STAT
	nCounter1	: EL3433Index := EL3433Index.listStart;
END_VAR

FOR nArrayIndex := TO_DWORD(EL3433Index.listStart) TO TO_DWORD(EL3433Index.listEnd) DO
	IF pstEL3433IO^.dIndex = ConstList.aEL3433Indices[nArrayIndex] THEN
		pTempReal := pstEL3433Data+nArrayIndex*SIZEOF(REAL);
		pTempReal^ := TO_REAL(pstEL3433IO^.dVariant) * ConstList.aEL3433IndicesScale[nArrayIndex];
		EXIT;
	END_IF
END_FOR

pstEL3433OutputIndex^ := ConstList.aEL3433Indices[nCounter1];
IF pstEL3433IO^.dIndex = ConstList.aEL3433Indices[nCounter1] THEN
	nCounter1 := nCounter1 + 1;
	IF nCounter1 > EL3433Index.listEnd THEN
		nCounter1 := EL3433Index.listStart;
	END_IF
END_IF

END_FUNCTION_BLOCK

// ---- POUs/CommunicationPrograms/BackgroundComm.TcPOU
PROGRAM BackgroundComm
VAR
END_VAR

HWVar.ModbusMaster();
HWVar.ModbusMaster1();

END_PROGRAM

// ---- POUs/MAIN.TcPOU
PROGRAM MAIN
VAR
	bInitDone : BOOL := FALSE;
	fml: FB_KL3208Config;
	KL3204Config1	:	FB_KL320xConfig;
	configCardIO: BOOL;
	readCardConfig: BOOL;
	iSensorType: INT;
END_VAR

IF NOT bInitDone THEN
	//GVL.bHV[1] := GVL.bLoadTank1;
	//GVL.bHV[2] := GVL.bLoadTank1;
	//GVL.bHV[4] := GVL.bLoadTank2;
	//GVL.bHV[5] := GVL.bLoadTank2;
	//GVL.bHV[7] := GVL.bLoadTank3;
	//GVL.bHV[8] := GVL.bLoadTank3;
	bInitDone := TRUE;
	
END_IF

IF GVL.fTE[4] < GVL.fTE[17] THEN
	// shut down pump 1 to precent heat loss
	//GVL.bP1 := FALSE;
	// start boiler to heat interal water
	
	ELSE 
	// open pump 1 to get heat from heat exchanger
	//GVL.bP1 := TRUE;
	// turn boiler on if necessary	
	
END_IF

ModbusCommunication();
CoolingFan();
//WaterFlowControl();
EnOcean_Dali();
BurningProcess();
ACT();  //setting up KL3204
//KL3208Config1(stindata:=hwvar.stKL3208_in, stOutData:=hwvar.stKL3208_out);

ACTION ACT:
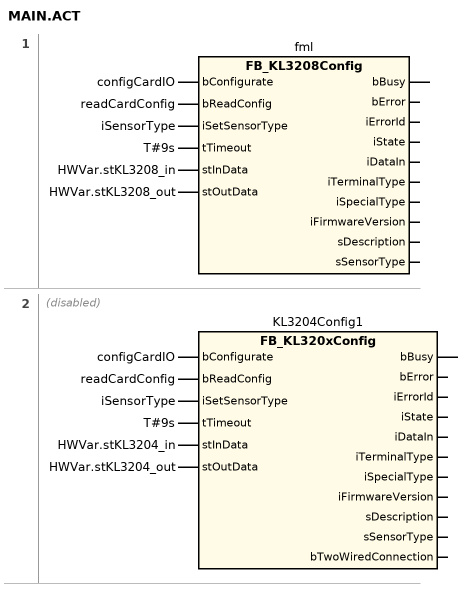
// NETWORK 1
fml(
    bConfigurate := configCardIO,
    bReadConfig := readCardConfig,
    iSetSensorType := iSensorType,
    tTimeout := T#9s,
    stInData := HWVar.stKL3208_in,
    stOutData := HWVar.stKL3208_out); // FB_KL3208Config

// NETWORK 2 (disabled)
// KL3204Config1(
//     bConfigurate := configCardIO,
//     bReadConfig := readCardConfig,
//     iSetSensorType := iSensorType,
//     tTimeout := T#9s,
//     stInData := HWVar.stKL3204_in,
//     stOutData := HWVar.stKL3204_out); // FB_KL320xConfig
END_ACTION

END_PROGRAM

// ---- POUs/ModbusCommunication.TcPOU
PROGRAM ModbusCommunication
VAR
	aP1, aP2, aP3			: ARRAY [GrundfosRegAddress.listStart +1 ..GrundfosRegAddress.listEnd -1] OF WORD;
	wMBData					: ARRAY [ATV212RegAddress.listStart +1 .. ATV212RegAddress.listEnd -1] OF WORD;
	nStep					: INT := 0;
	wP1Control, wP2Control, wP3Control	: ARRAY [100..105] OF WORD := [
		16#0000,
		16#0080,
		0,
		0,
		0,
		600
	];
	wFeederControl			: ARRAY [16#FA00..16#FA01] OF WORD := [];
	wFeederControlAddress	: WORD;
	wP1Status, wP2Status, wP3Status	: ARRAY[200..220] OF WORD;
	wFeederStatus			: ARRAY[16#D01..16#E01] OF WORD;
	wContent				: WORD;
END_VAR

VAR CONSTANT
	bP1Addr					: BYTE := 2;
	bP2Addr					: BYTE := 4;
	bP3Addr					: BYTE := 6;
	bFeederAddr				: BYTE := 5;
	wStartPumpCmd			: WORD := 16#0027; //27
	wStopPumpCmd			: WORD := 16#0025; //25
END_VAR

HWVar.ModbusMaster.ReadRegs(Execute := FALSE);
HWVar.ModbusMaster.WriteRegs(Execute := FALSE);
HWVar.ModbusMaster1.ReadRegs(Execute := FALSE);
HWVar.ModbusMaster1.WriteRegs(Execute := FALSE);
IF GVL.bP1 THEN
               wP1Control[100] := wStartPumpCmd;
ELSE 
               wP1Control[100] := wStopPumpCmd;
END_IF
IF GVL.bP2 THEN
               wP2Control[100] := wStartPumpCmd;
ELSE 
               wP2Control[100] := wStopPumpCmd;
END_IF
IF GVL.bP3 THEN
               wP3Control[100] := wStartPumpCmd;
ELSE 
               wP3Control[100] := wStopPumpCmd;
END_IF

CASE nStep OF 
	0: 
		P1Read(); 
    1: 
        P2Read(); 
    2: 
        GrundfosDataConversion(arrReg:= aP1, pstGrundfosMagna3:= ADR(GVL.stP1)); 
        GrundfosDataConversion(arrReg:= aP2, pstGrundfosMagna3:= ADR(GVL.stP2));
        nStep := 3;
    3:
        P1Write();
    4:
        P2Write();
    5:
        P1ReadStatus();
    6:
        P2ReadStatus();
    7:
        FeederReadSingle();
    8:
        ATV212DataConversion(arrReg := wMBData, pstATV212 := ADR(GVL.stFeeder));
        nStep := 9;
    9:
        FeederControlRun();
	10: 
		FeederSpeedControl(wContent => wContent);
		FeederWrite(wContent, 16#FA01);
    11:
        FeederStatus();
        //nStep := 0;
	12:
		P3Read();
	13:
		GrundfosDataConversion(arrReg:= aP3, pstGrundfosMagna3:= ADR(GVL.stP3)); 
		nStep := 14;
	14:
		P3Write();
	15:
		P3ReadStatus();
END_CASE;

METHOD ATV212DataConversion : BOOL
VAR_INPUT
               arrReg   : ARRAY [ATV212RegAddress.listStart +1 .. ATV212RegAddress.listEnd -1] OF WORD;
               pstATV212           : POINTER TO ATV212;
END_VAR

VAR
			// iMemIndex: ATV212RegAddress;
			iMemIndex: WORD := ATV212RegAddress.listStart +1;
               a_MbRegValue  : ARRAY [ATV212RegAddress.listStart +1 .. ATV212RegAddress.listEnd -1] OF REAL;
END_VAR
WHILE (iMemIndex <=  ATV212RegAddress.listEnd) DO
	a_MbRegValue[iMemIndex] := (arrReg[iMemIndex])*Scale.fATV212Scale[iMemIndex];
    iMemIndex := iMemIndex + 1;
END_WHILE
MEMCPY(pstATV212, ADR(a_MbRegValue), SIZEOF(ATV212));
END_METHOD

METHOD FeederControlRun : BOOL
VAR_INPUT
END_VAR

VAR
	fbStartStop: RS;
	reStart: R_TRIG;
	wContent: WORD;
	wAddress: WORD;
	tmFeederOn: TON;
END_VAR
wAddress := 16#FA00;

IF GVL.stFeederControl.bStart THEN
	IF gvl.stFeederControl.bForward THEN
		wContent := 16#C400;
		ELSE wContent := 16#C600;
	END_IF
	FeederWrite(wContent, wAddress);
ELSE
	wContent := 16#C000;
	gvl.stFeederControl.fFrequency := 0;
	FeederWrite(wContent, wAddress);
END_IF
END_METHOD

METHOD FeederReadSingle : BOOL
VAR_INPUT
END_VAR
IF (NOT HWVar.ModbusMaster.BUSY) THEN
	HWVar.ModbusMaster.ReadRegs(
		UnitID := bFeederAddr,
		Quantity := 4,
		MBAddr := 16#1875,
		cbLength := SIZEOF(wMBData),
		pMemoryAddr := ADR(wMBData),
		Execute := TRUE,
		Timeout := T#5S,
		BUSY => ,
		Error =>
		);
		nStep := 8;
END_IF;
END_METHOD

METHOD FeederStatus : BOOL
VAR_INPUT

END_VAR
IF (NOT HWVar.ModbusMaster.BUSY) THEN
	HWVar.ModbusMaster.ReadRegs(
		UnitID := bFeederAddr,
		Quantity := 1,
		MBAddr := 16#FD00,
		cbLength := SIZEOF(wFeederStatus),
		pMemoryAddr := ADR(wFeederStatus),
		Execute := TRUE,
		Timeout := T#5S,
		BUSY => ,
		Error =>
		);
		nStep := 12;
END_IF;
END_METHOD

METHOD FeederWrite : BOOL
VAR_INPUT
	wFeederControl: WORD;
	wFeederControlAddress: WORD;
END_VAR
IF (NOT HWVar.ModbusMaster.BUSY) THEN
	HWVar.ModbusMaster.WriteRegs(
		UnitID := bFeederAddr,
		Quantity := 1,
		MBAddr := wFeederControlAddress,
		cbLength := SIZEOF(WORD),
		pMemoryAddr := ADR(wFeederControl),
		Execute := TRUE,
		Timeout := T#5S,
		BUSY => ,
		Error =>
		);	
	nStep := nStep+1;	
END_IF;
END_METHOD

METHOD PUBLIC GrundfosDataConversion : BOOL
VAR_INPUT
	arrReg	: ARRAY [GrundfosRegAddress.listStart +1 ..GrundfosRegAddress.listEnd -1] OF WORD;
	pstGrundfosMagna3	: POINTER TO GrundfosMagna3;
END_VAR

VAR
	iMemIndex: WORD := GrundfosRegAddress.listStart +1;
	iRegIndex: WORD := GrundfosRegAddress.listStart +1;
	a_MbRegValue	: ARRAY [300..350] OF REAL;
	dwMergedReg		: DWORD;
END_VAR
WHILE (iMemIndex <  GrundfosRegAddress.listEnd AND iRegIndex < 351) DO
	IF (iRegIndex <> 311) 
		AND (iRegIndex <> 326)
		AND (iRegIndex <> 328) 
		AND (iRegIndex <> 331)
		AND (iRegIndex <> 333)
		AND (iRegIndex <> 342)
		AND (iRegIndex <> 351)
		AND (iRegIndex <> 353)
		AND (iRegIndex <> 356)
		AND (iRegIndex <> 358)
		AND (iRegIndex <> 360) THEN
		a_MbRegValue[iRegIndex] := (arrReg[iMemIndex])*Scale.fGrundfosScale[iRegIndex];
		iMemIndex := iMemIndex + 1;
		iRegIndex := iRegIndex + 1;
	ELSE
		dwMergedReg := SHL(WORD_TO_DWORD(arrReg[iMemIndex]),16) OR WORD_TO_DWORD(arrReg[iMemIndex+1]);
		a_MbRegValue[iRegIndex] := (DWORD_TO_REAL(dwMergedReg))*Scale.fGrundfosScale[iRegIndex];
		iMemIndex := iMemIndex + 2;
		iRegIndex := iRegIndex + 1;
	END_IF
END_WHILE
MEMCPY(pstGrundfosMagna3, ADR(a_MbRegValue), SIZEOF(GrundfosMagna3));
END_METHOD

METHOD PRIVATE P1Read : BOOL
VAR_STAT
	nRegisterAddress	: GrundfosRegAddress;
END_VAR
IF (NOT HWVar.ModbusMaster.BUSY) THEN
	HWVar.ModbusMaster.ReadRegs(
		UnitID := bP1Addr,
		Quantity := 61,
		MBAddr := 300,
		cbLength := SIZEOF(aP1),
		pMemoryAddr := ADR(aP1),
		Execute := TRUE,
		Timeout := T#5S,
		BUSY => ,
		Error =>
		);
		nStep := 1;
END_IF;
END_METHOD

METHOD PRIVATE P1ReadStatus : BOOL
VAR_STAT
	nRegisterAddress	: GrundfosRegAddress;
END_VAR
IF (NOT HWVar.ModbusMaster.BUSY) THEN
	HWVar.ModbusMaster.ReadRegs(
		UnitID := bP1Addr,
		Quantity := 21,
		MBAddr := 200,
		cbLength := SIZEOF(wP1Status),
		pMemoryAddr := ADR(wP1Status),
		Execute := TRUE,
		Timeout := T#5S,
		BUSY => ,
		Error =>
		);
		nStep := 6;
END_IF;
END_METHOD

METHOD PRIVATE P1Write : BOOL
VAR_STAT
	nRegisterAddress	: GrundfosRegAddress;
END_VAR
IF (NOT HWVar.ModbusMaster.BUSY) THEN
	HWVar.ModbusMaster.WriteRegs(
		UnitID := bP1Addr,
		Quantity := 6,
		MBAddr := 100,
		cbLength := SIZEOF(wP1Control),
		pMemoryAddr := ADR(wP1Control),
		Execute := TRUE,
		Timeout := T#5S,
		BUSY => ,
		Error =>
		);
		nStep := 4;
END_IF;
END_METHOD

METHOD PRIVATE P2Read : BOOL
VAR_STAT
	nRegisterAddress	: GrundfosRegAddress;
END_VAR
IF (NOT HWVar.ModbusMaster.BUSY) THEN
	HWVar.ModbusMaster.ReadRegs(
		UnitID := bP2Addr,
		Quantity := 61,
		MBAddr := 300,
		cbLength := SIZEOF(aP2),
		pMemoryAddr := ADR(aP2),
		Execute := TRUE,
		Timeout := T#5S,
		BUSY => ,
		Error =>
		);
		nStep := 2;
END_IF;
END_METHOD

METHOD PRIVATE P2ReadStatus : BOOL
VAR_STAT
	nRegisterAddress	: GrundfosRegAddress;
END_VAR
IF (NOT HWVar.ModbusMaster.BUSY) THEN
	HWVar.ModbusMaster.ReadRegs(
		UnitID := bP2Addr,
		Quantity := 21,
		MBAddr := 200,
		cbLength := SIZEOF(wP2Status),
		pMemoryAddr := ADR(wP2Status),
		Execute := TRUE,
		Timeout := T#5S,
		BUSY => ,
		Error =>
		);
		nStep := 7;
END_IF;
END_METHOD

METHOD PRIVATE P2Write : BOOL
VAR_STAT
	nRegisterAddress	: GrundfosRegAddress;
END_VAR
IF (NOT HWVar.ModbusMaster.BUSY) THEN
	HWVar.ModbusMaster.WriteRegs(
		UnitID := bP2Addr,
		Quantity := 6,
		MBAddr := 100,
		cbLength := SIZEOF(wP2Control),
		pMemoryAddr := ADR(wP2Control),
		Execute := TRUE,
		Timeout := T#5S,
		BUSY => ,
		Error =>
		);
		nStep := 5;
END_IF;
END_METHOD

METHOD P3Read : BOOL
VAR_INPUT
END_VAR

VAR

END_VAR
IF (NOT HWVar.ModbusMaster1.BUSY) THEN
	HWVar.ModbusMaster1.ReadRegs(
		UnitID := bP3Addr,
		Quantity := 61,
		MBAddr := 300,
		cbLength := SIZEOF(aP3),
		pMemoryAddr := ADR(aP3),
		Execute := TRUE,
		Timeout := T#5S,
		BUSY => ,
		Error =>
		);
		nStep := 13;
END_IF;
END_METHOD

METHOD P3ReadStatus : BOOL
VAR_INPUT
END_VAR
IF (NOT HWVar.ModbusMaster1.BUSY) THEN
	HWVar.ModbusMaster1.ReadRegs(
		UnitID := bP3Addr,
		Quantity := 21,
		MBAddr := 200,
		cbLength := SIZEOF(wP3Status),
		pMemoryAddr := ADR(wP3Status),
		Execute := TRUE,
		Timeout := T#5S,
		BUSY => ,
		Error =>
		);
		nStep := 0;
END_IF;
END_METHOD

METHOD P3Write : BOOL
VAR_INPUT
END_VAR
IF (NOT HWVar.ModbusMaster1.BUSY) THEN
	HWVar.ModbusMaster1.WriteRegs(
		UnitID := bP3Addr,
		Quantity := 6,
		MBAddr := 100,
		cbLength := SIZEOF(wP3Control),
		pMemoryAddr := ADR(wP3Control),
		Execute := TRUE,
		Timeout := T#5S,
		BUSY => ,
		Error =>
		);
		nStep := 15;
END_IF;
END_METHOD

ACTION SC01Read:
nStep := 3;
END_ACTION

END_PROGRAM

// ---- POUs/BurningProcess/FeederSpeedControl.TcPOU
PROGRAM FeederSpeedControl
VAR
	FeederMode: INT;
	fbMaximumSpeed			: FB_OnOffTimer;
	fbMinimumSpeed			: FB_OnOffTimer;
	fbManualSpeed			: FB_OnOffTimer;
END_VAR

VAR_OUTPUT
	wContent: WORD;
END_VAR

IF GVL.stFeederControl.bManual THEN
	FeederMode := 2;
	ELSE IF GVL.fTE[17] > ConstList.WaterTempMax THEN
			FeederMode := 1;
			ELSE IF GVL.fTE[17] < ConstList.WaterTempMin THEN 
				FeederMode := 0;
			END_IF
	END_IF
END_IF

CASE FeederMode OF
	0:
		// Maximum speed
		fbMaximumSpeed(tTimeOn := T#4S, tTimeOff := T#25S, nSpeedOn := 2500, nSpeedOff := 0000, nSpeedOut => wContent);
	1:
		// Stand-by speed	
		fbMaximumSpeed(tTimeOn := T#3.25S, tTimeOff := T#12M30S, nSpeedOn := 2500, nSpeedOff := 0000, nSpeedOut => wContent);
	2:
		// Manual mode
		fbManualSpeed(tTimeOn := gvl.stFeederControl.tTimeOn, tTimeOff := gvl.stFeederControl.tTimeOff, nSpeedOn := REAL_TO_WORD(GVL.stFeederControl.fFrequency*100), nSpeedOff := 0000, nSpeedOut => wContent);
END_CASE

IF gvl.stFeederControl.bStart AND gvl.stFeederControl.bForward THEN // not set non-zero freq if motor's not on
	//gvl.stFeederControl.fFrequency := WORD_TO_REAL(wContent/100); // update current freq
	ELSE wContent := 0000;
		gvl.stFeederControl.fFrequency := 0;
END_IF

END_PROGRAM

// ---- POUs/EnergyFlow/CoolingFan.TcPOU
PROGRAM CoolingFan
VAR
	bLowFlowTempWarning : BOOL := FALSE;
	bUnloadBoilerToTanks : BOOL := FALSE;
	tonPump2: TON;
END_VAR

// Automatic controll for lauhdutin fan
// Turn fan OFF if in-out temp diff > 10 or out temp < 55 
IF GVL.fTE[15]-GVL.fTE[16] > 10 THEN 
	GVL.bFanPower := FALSE; 
ELSE 
	IF NOT bLowFlowTempWarning THEN
		GVL.bFanPower := TRUE;
	END_IF
END_IF
IF GVL.fTE[15] < 55 THEN // activate low flow temp warning
	bLowFlowTempWarning := TRUE;
	GVL.bFanPower := FALSE;
	GVL.bP3 := FALSE;
	GVL.bHV[11] := FALSE;
END_IF
IF GVl.fTE[15] > 56 THEN
	GVL.bP3 := TRUE;;
	GVL.bHV[11] := TRUE;
END_IF
IF GVL.fTE[15] > 59 THEN  // reset low flow temp warning
	bLowFlowTempWarning := FALSE;
END_IF

END_PROGRAM

// ---- POUs/Lights/EnOcean_Dali.TcPOU
PROGRAM EnOcean_Dali
VAR
	fbKL6581	: FB_KL6581;
	dwID		: DWORD;
	bReady		: BOOL;
	bBusy		: BOOL;
	bError		: BOOL;
	iErrorID	: INT;
	EnOceanID 	: DWORD;
	EnOceanAction : BYTE;
	
	// These are in globals
	// st6581_in	: KL6581_Input;
	// st6581_out	: KL6581_Output;
	// stKL6581	: STR_KL6581;
	
	bLeftButtonUp	: BOOL;
	bLeftButtonDown	: BOOL;
	bRightButtonUp	: BOOL;
	bRightButtonDown: BOOL;
	
	TankLight	: FB_DALIV2Dimmer1Switch; //left button
	BoilerLight	: FB_DALIV2Dimmer1Switch; //right button
	DaliAddressing	: FB_DALIV2AddressingIntRandomAddressing;
	DaliSearch		: FB_DALIV2SearchAddr;
	
	bDaliBusy	: BOOL;
	bDaliError	: BOOL;
	nDaliErrorId: UDINT;
	
	bStart : BOOL;
	nAddressedDevices: BYTE;
	fbTankLightTimer: TON;
	nTankLightDim: BYTE;
	nBoilerLightDim: BYTE;
	fbBoilerLightTimer: TON;
	fbTankLightOff: TON;
	fbBoilerLightOff: TON;
END_VAR

fbTankLightTimer(IN:= , PT:= T#45M, Q=> , ET=> );
fbBoilerLightTimer(IN:= , PT:= T#45M, Q=> , ET=> );
fbTankLightOff(IN:= , PT:= T#2M, Q=> , ET=> );
fbBoilerLightOff(IN:= , PT:= T#2M, Q=> , ET=> );
fbKL6581(
	bInit := TRUE, 
	nIdx := 7, 
	bReady => bReady, 
	bBusy => bBusy, 
	bError => bError, 
	iErrorID => iErrorID, 
	str_KL6581 => HWVar.stKL6581, 
	stKL6581_in := HWVar.st6581_in , 
	stKL6581_out := HWvar.st6581_out);
	
EnOceanID := HWVar.stKL6581.dw_ID;
EnOceanAction := HWVar.stKL6581.ar_DB[3]; 

IF (EnOceanAction = 16#30) THEN 
	bLeftButtonUp := TRUE; fbTankLightTimer.IN := TRUE; nTankLightDim := 254; fbTankLightOff.IN := FALSE; ELSE bLeftButtonUp := FALSE;
END_IF
IF (EnOceanAction = 16#10) THEN 
	bLeftButtonDown := TRUE; ELSE bLeftButtonDown := FALSE;
END_IF
IF (EnOceanAction = 16#70) THEN 
	bRightButtonUp := TRUE; fbBoilerLightTimer.IN := TRUE; nBoilerLightDim := 254; fbBoilerLightOff.IN := FALSE; ELSE bRightButtonUp := FALSE;
END_IF
IF (EnOceanAction = 16#50) THEN 
	bRightButtonDown := TRUE; ELSE bRightButtonDown := FALSE;
END_IF

IF fbTankLightTimer.Q THEN
	nTankLightDim := 170;
	fbTankLightTimer.IN := FALSE;
	fbTankLightOff.IN := TRUE;
END_IF

IF fbTankLightOff.Q THEN
	nTankLightDim := 0;
	fbTankLightOff.IN := FALSE;
END_IF

IF fbBoilerLightTimer.Q THEN
	nBoilerLightDim := 170;
	fbBoilerLightTimer.IN := FALSE;
	fbBoilerLightOff.IN := TRUE;
END_IF

IF fbBoilerLightOff.Q THEN
	nBoilerLightDim := 0;
	fbBoilerLightOff.IN := FALSE;
END_IF

TankLight(
	bSwitchDimm:= bLeftButtonUp, 
	bOn:= bLeftButtonUp, 
	bOff:= bLeftButtonDown, 
	bSetDimmValue:= bLeftButtonUp, 
	nDimmValue:= nTankLightDim, 
	tSwitchOverTime:= T#50MS, 
	tCycleDelay:= T#500MS, 
	bMemoryModeOn:= FALSE, 
	nOnValueWithoutMemoryMode:= 254, // max value
	nAddr:= 0, 
	eAddrType:= , 
	nMasterDevAddr:= , // addr of master dev in group, not used for now
	nMinLevelMasterDev:= 126, // min value
	nMaxLevelMasterDev:= 254, //max value
	tCycleActualLevelMasterDev:= , 
	nActualLevelMasterDev=> , 
	bBusy=> bDaliBusy, 
	bError=> bDaliError, 
	nErrorId=> nDaliErrorId, 
	stCommandBuffer:= HWVar.stKL6811_CommandBuffer);

BoilerLight(
	bSwitchDimm:= bRightButtonUp, 
	bOn:= bRightButtonUp, 
	bOff:= bRightButtonDown, 
	bSetDimmValue:= bRightButtonUp, 
	nDimmValue:= nBoilerLightDim, 
	tSwitchOverTime:= T#50MS, 
	tCycleDelay:= T#500MS, 
	bMemoryModeOn:= FALSE, 
	nOnValueWithoutMemoryMode:= 254, // max value
	nAddr:= 1, 
	eAddrType:= , 
	nMasterDevAddr:= , // addr of master dev in group, not used for now
	nMinLevelMasterDev:= 126, // min value
	nMaxLevelMasterDev:= 254, //max value
	tCycleActualLevelMasterDev:= , 
	nActualLevelMasterDev=> , 
	bBusy=> bDaliBusy, 
	bError=> bDaliError, 
	nErrorId=> nDaliErrorId, 
	stCommandBuffer:= HWVar.stKL6811_CommandBuffer);

END_PROGRAM

// ---- POUs/BurningProcess/BurningProcess.TcPOU
PROGRAM BurningProcess
VAR

END_VAR

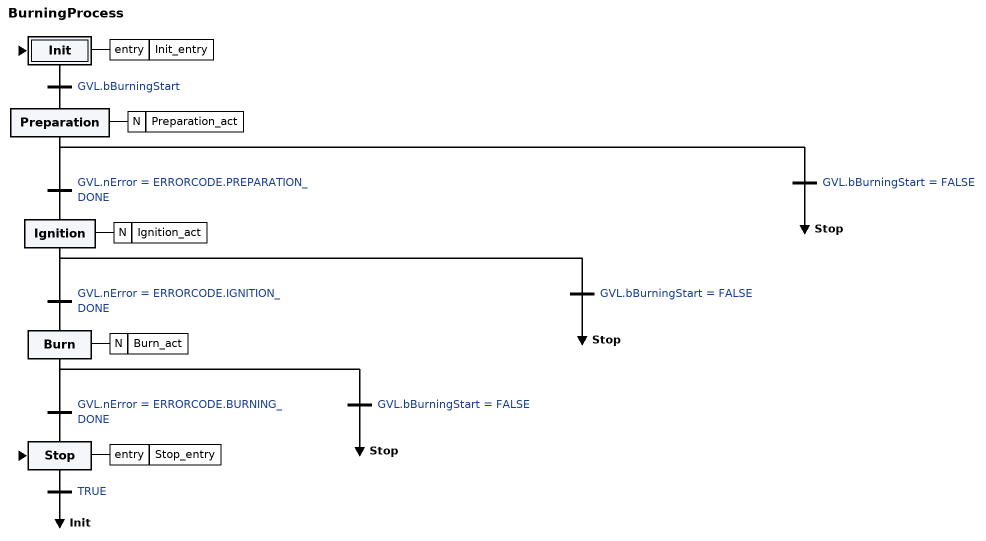
INITIAL_STEP Init:
    Init_entry(P1);  // entry action
END_STEP
TRANSITION FROM Init TO Preparation
    := GVL.bBurningStart;
END_TRANSITION
STEP Preparation:
    Preparation_act(N);
END_STEP
TRANSITION FROM Preparation TO Ignition
    := GVL.nError = ERRORCODE.PREPARATION_DONE;
END_TRANSITION
STEP Ignition:
    Ignition_act(N);
END_STEP
TRANSITION FROM Ignition TO Burn
    := GVL.nError = ERRORCODE.IGNITION_DONE;
END_TRANSITION
STEP Burn:
    Burn_act(N);
END_STEP
TRANSITION FROM Burn TO Stop
    := GVL.nError = ERRORCODE.BURNING_DONE;
END_TRANSITION
TRANSITION FROM Burn TO Stop
    := GVL.bBurningStart = FALSE;
END_TRANSITION
TRANSITION FROM Ignition TO Stop
    := GVL.bBurningStart = FALSE;
END_TRANSITION
TRANSITION FROM Preparation TO Stop
    := GVL.bBurningStart = FALSE;
END_TRANSITION
STEP Stop:
    Stop_entry(P1);  // entry action
END_STEP
TRANSITION FROM Stop TO Init
    := TRUE;
END_TRANSITION

ACTION Burn_act:
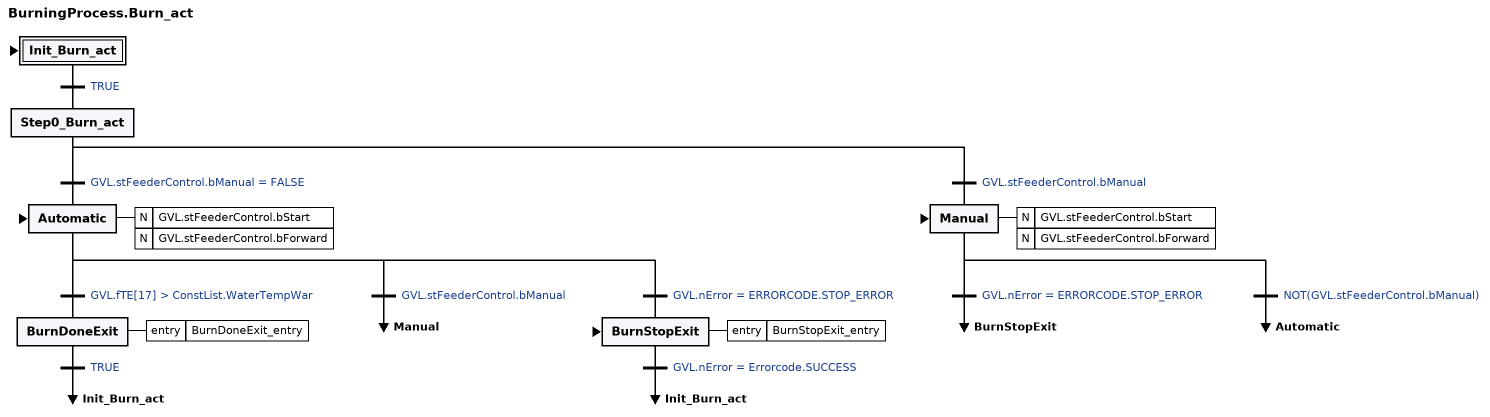
INITIAL_STEP Init_Burn_act:
END_STEP
TRANSITION FROM Init_Burn_act TO Step0_Burn_act
    := TRUE;
END_TRANSITION
STEP Step0_Burn_act:
END_STEP
TRANSITION FROM Step0_Burn_act TO Automatic
    := GVL.stFeederControl.bManual = FALSE;
END_TRANSITION
STEP Automatic:
    GVL.stFeederControl.bStart(N);
    GVL.stFeederControl.bForward(N);
END_STEP
TRANSITION FROM Automatic TO BurnDoneExit
    := GVL.fTE[17] > ConstList.WaterTempWar;
END_TRANSITION
STEP BurnDoneExit:
    BurnDoneExit_entry(P1);  // entry action
END_STEP
TRANSITION FROM BurnDoneExit TO Init_Burn_act
    := TRUE;
END_TRANSITION
TRANSITION FROM Automatic TO Manual
    := GVL.stFeederControl.bManual;
END_TRANSITION
TRANSITION FROM Automatic TO BurnStopExit
    := GVL.nError = ERRORCODE.STOP_ERROR;
END_TRANSITION
STEP BurnStopExit:
    BurnStopExit_entry(P1);  // entry action
END_STEP
TRANSITION FROM BurnStopExit TO Init_Burn_act
    := GVL.nError = Errorcode.SUCCESS;
END_TRANSITION
TRANSITION FROM Step0_Burn_act TO Manual
    := GVL.stFeederControl.bManual;
END_TRANSITION
STEP Manual:
    GVL.stFeederControl.bStart(N);
    GVL.stFeederControl.bForward(N);
END_STEP
TRANSITION FROM Manual TO BurnStopExit
    := GVL.nError = ERRORCODE.STOP_ERROR;
END_TRANSITION
TRANSITION FROM Manual TO Automatic
    := NOT(GVL.stFeederControl.bManual);
END_TRANSITION
// branch label Branch1_Burn_act
// branch label Branch2_Burn_act
// branch label Branch0_Burn_act
END_ACTION

ACTION BurnDoneExit_entry:
GVL.nError := ERRORCODE.BURNING_DONE;
END_ACTION

ACTION BurnStopExit_entry:
GVL.nError := errorcode.STOP_ERROR;
END_ACTION

ACTION ClearGases_active:
GVL.stPrimaryFan.nSpeed := 100;
GVL.stSecondaryFan.nSpeed := 100;
END_ACTION

ACTION ClearGases_exit:
GVL.stPrimaryFan.nSpeed := 25;
GVL.stSecondaryFan.nSpeed := 25;
END_ACTION

ACTION FanControl_act:
IF	GVL.fO2 > 10 THEN
	GVL.stPrimaryFan.nSpeed := 25;
	ELSE IF GVL.fO2 < 6 THEN
		GVL.stPrimaryFan.nSpeed := 50;
	END_IF
END_IF
END_ACTION

ACTION FeederOn_active:
GVL.stFeederControl.bStart := TRUE;
GVL.stFeederControl.bForward := TRUE;
GVL.stFeederControl.bManual := TRUE;
GVL.stFeederControl.fFrequency := 25;
GVL.stFeederControl.tTimeOn := T#10S; // 100s
GVL.stFeederControl.tTimeOff := T#0S;
END_ACTION

ACTION FeederOn_exit:
GVL.stFeederControl.bStart := FALSE;
GVL.stFeederControl.bForward := FALSE;
GVL.stFeederControl.bManual := FALSE;
GVL.nError := Errorcode.PREPARATION_DONE;
END_ACTION

ACTION FlameDetected_entry:
GVL.nError := ERRORCODE.PREPARATION_FLAME;
END_ACTION

ACTION Ignite_active:
GVL.stFI1.bBlower := TRUE;
GVL.stFI1.bHeating := TRUE;
END_ACTION

ACTION Ignition_act:
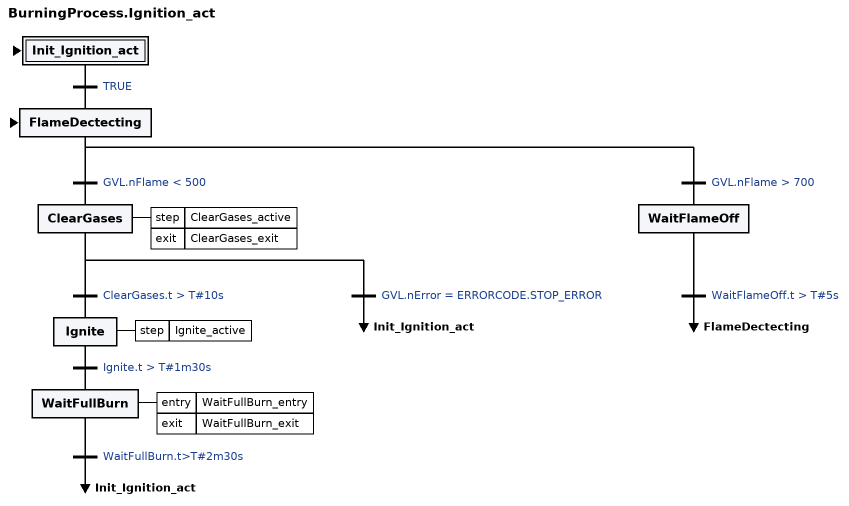
INITIAL_STEP Init_Ignition_act:
END_STEP
TRANSITION FROM Init_Ignition_act TO FlameDectecting
    := TRUE;
END_TRANSITION
STEP FlameDectecting:
END_STEP
TRANSITION FROM FlameDectecting TO ClearGases
    := GVL.nFlame < 500;
END_TRANSITION
STEP ClearGases:
    ClearGases_active(N);  // step action
    ClearGases_exit(P0);  // exit action
END_STEP
TRANSITION FROM ClearGases TO Ignite
    := ClearGases.t > T#10s;
END_TRANSITION
STEP Ignite:
    Ignite_active(N);  // step action
END_STEP
TRANSITION FROM Ignite TO WaitFullBurn
    := Ignite.t > T#1m30s;
END_TRANSITION
STEP WaitFullBurn:
    WaitFullBurn_entry(P1);  // entry action
    WaitFullBurn_exit(P0);  // exit action
END_STEP
TRANSITION FROM WaitFullBurn TO Init_Ignition_act
    := WaitFullBurn.t>T#2m30s;
END_TRANSITION
TRANSITION FROM ClearGases TO Init_Ignition_act
    := GVL.nError = ERRORCODE.STOP_ERROR;
END_TRANSITION
TRANSITION FROM FlameDectecting TO WaitFlameOff
    := GVL.nFlame > 700;
END_TRANSITION
STEP WaitFlameOff:
END_STEP
TRANSITION FROM WaitFlameOff TO FlameDectecting
    := WaitFlameOff.t > T#5s;
END_TRANSITION
// branch label Branch1_Ignition_act
// branch label Branch0_Ignition_act
END_ACTION

ACTION Init_entry:
GVL.stPrimaryFan.nSpeed := 0;
GVL.stSecondaryFan.nSpeed := 0;
GVL.stFeederControl.bStart := FALSE;
GVL.stFeederControl.bForward := FALSE;
GVL.nError := 0;
END_ACTION

ACTION Preparation_act:
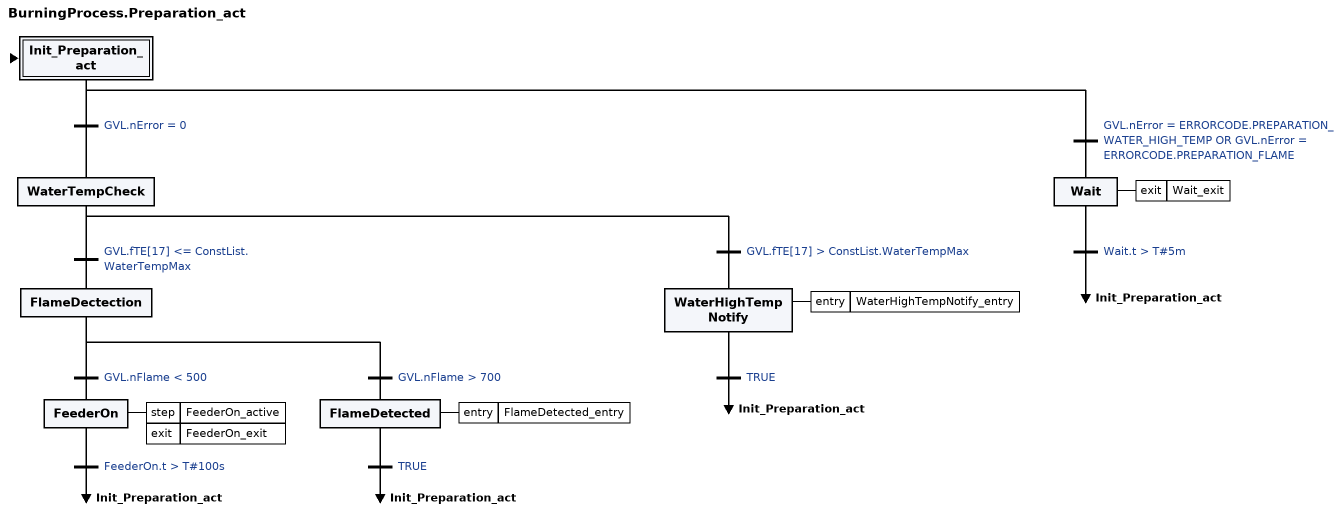
INITIAL_STEP Init_Preparation_act:
END_STEP
TRANSITION FROM Init_Preparation_act TO WaterTempCheck
    := GVL.nError = 0;
END_TRANSITION
TRANSITION FROM Init_Preparation_act TO Wait
    := GVL.nError = ERRORCODE.PREPARATION_WATER_HIGH_TEMP OR GVL.nError = ERRORCODE.PREPARATION_FLAME;
END_TRANSITION
STEP Wait:
    Wait_exit(P0);  // exit action
END_STEP
TRANSITION FROM Wait TO Init_Preparation_act
    := Wait.t > T#5m;
END_TRANSITION
STEP WaterTempCheck:
END_STEP
TRANSITION FROM WaterTempCheck TO FlameDectection
    := GVL.fTE[17] <= ConstList.WaterTempMax;
END_TRANSITION
STEP FlameDectection:
END_STEP
TRANSITION FROM FlameDectection TO FeederOn
    := GVL.nFlame < 500;
END_TRANSITION
STEP FeederOn:
    FeederOn_active(N);  // step action
    FeederOn_exit(P0);  // exit action
END_STEP
TRANSITION FROM FeederOn TO Init_Preparation_act
    := FeederOn.t > T#100s;
END_TRANSITION
TRANSITION FROM FlameDectection TO FlameDetected
    := GVL.nFlame > 700;
END_TRANSITION
STEP FlameDetected:
    FlameDetected_entry(P1);  // entry action
END_STEP
TRANSITION FROM FlameDetected TO Init_Preparation_act
    := TRUE;
END_TRANSITION
TRANSITION FROM WaterTempCheck TO WaterHighTempNotify
    := GVL.fTE[17] > ConstList.WaterTempMax;
END_TRANSITION
STEP WaterHighTempNotify:
    WaterHighTempNotify_entry(P1);  // entry action
END_STEP
TRANSITION FROM WaterHighTempNotify TO Init_Preparation_act
    := TRUE;
END_TRANSITION
// branch label Branch2_Preparation_act
// branch label Branch1_Preparation_act
// branch label Branch0_Preparation_act
END_ACTION

ACTION Stop_entry:
GVL.bBurningStart := FALSE;
GVL.stPrimaryFan.nSpeed := 0;
GVL.stSecondaryFan.nSpeed := 0;
GVL.stFeederControl.bStart := FALSE;
GVL.stFeederControl.bForward := FALSE;
GVL.stFI1.bHeating := FALSE;
GVL.stFI1.bBlower := FALSE;
GVL.nError := 0;
//GVL.bP1 := FALSE;
//GVL.bP2 := FALSE;
END_ACTION

ACTION Wait_exit:
GVL.nError := ERRORCODE.SUCCESS;
END_ACTION

ACTION WaitFullBurn_entry:
GVL.stPrimaryFan.nSpeed := 35;
GVL.stFI1.bHeating := FALSE;
END_ACTION

ACTION WaitFullBurn_exit:
GVL.stFI1.bBlower := FALSE;
GVL.nError := ERRORCODE.IGNITION_DONE;
END_ACTION

ACTION WaterHighTempNotify_entry:
GVL.nError := ERRorcode.PREPARATION_WATER_HIGH_TEMP;
END_ACTION

END_PROGRAM

// ---- POUs/EnergyFlow/WaterFlowControl.TcPOU
PROGRAM WaterFlowControl
VAR
END_VAR

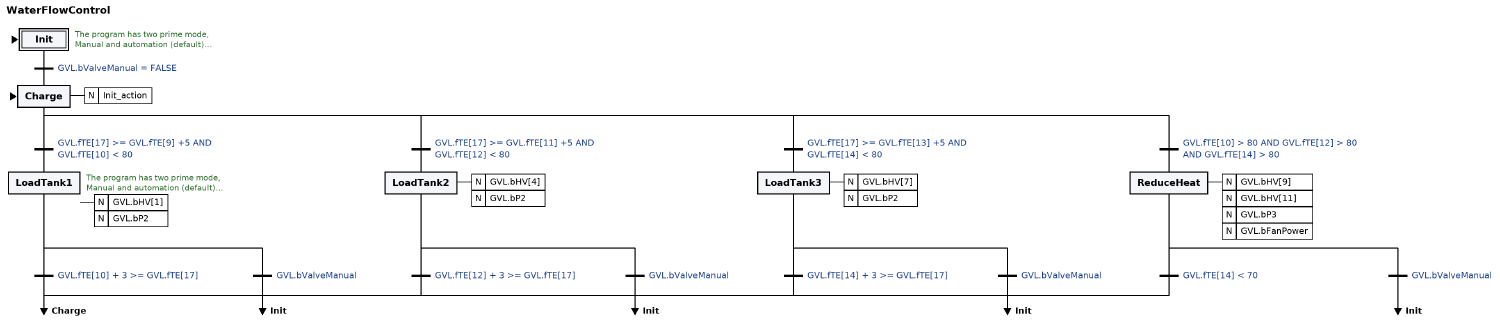
// The program has two prime mode, Manual and automation (default). Manual mode counteracts the whole program so that you can control flows as you want. In automation mode, if boiler water temperature is at least 5 degree greater than tank water's, and tank water is lower than 80 degree; valve and pump will be turned on to load water to tank. If more than one tank meet the requirements, the loading process order will be 1,2,3. There's always one tank being loaded at a time. If 3 tanks have above 80 degree temperature, pump 3 and corresponding valves will be opened to unload the heat. If tank temperature is greater than boiler's, loading will stop in order to avoid heat loss. Consider having most critical condition/function on the most left branches, because in alternative branches, the order is from left to right.
INITIAL_STEP Init:
END_STEP
TRANSITION FROM Init TO Charge
    := GVL.bValveManual = FALSE;
END_TRANSITION
STEP Charge:
    Init_action(N);
END_STEP
TRANSITION FROM Charge TO LoadTank1
    := GVL.fTE[17] >= GVL.fTE[9] +5 AND GVL.fTE[10] < 80;
END_TRANSITION
// The program has two prime mode, Manual and automation (default). Manual mode counteracts the whole program so that you can control flows as you want. In automation mode, if boiler water temperature is at least 5 degree greater than tank water's, and tank water is lower than 80 degree; valve and pump will be turned on to load water to tank. If more than one tank meet the requirements, the loading process order will be 1,2,3. There's always one tank being loaded at a time. If 3 tanks have above 80 degree temperature, pump 3 and corresponding valves will be opened to unload the heat. If tank temperature is greater than boiler's, loading will stop in order to avoid heat loss. Consider having most critical condition/function on the most left branches, because in alternative branches, the order is from left to right.
STEP LoadTank1:
    GVL.bHV[1](N);
    GVL.bP2(N);
END_STEP
TRANSITION FROM LoadTank1 TO Charge
    := GVL.fTE[10] + 3 >= GVL.fTE[17];
END_TRANSITION
TRANSITION FROM LoadTank1 TO Init
    := GVL.bValveManual;
END_TRANSITION
TRANSITION FROM Charge TO LoadTank2
    := GVL.fTE[17] >= GVL.fTE[11] +5 AND GVL.fTE[12] < 80;
END_TRANSITION
STEP LoadTank2:
    GVL.bHV[4](N);
    GVL.bP2(N);
END_STEP
TRANSITION FROM LoadTank2 TO Charge
    := GVL.fTE[12] + 3 >= GVL.fTE[17];
END_TRANSITION
TRANSITION FROM LoadTank2 TO Init
    := GVL.bValveManual;
END_TRANSITION
TRANSITION FROM Charge TO LoadTank3
    := GVL.fTE[17] >= GVL.fTE[13] +5 AND GVL.fTE[14] < 80;
END_TRANSITION
STEP LoadTank3:
    GVL.bHV[7](N);
    GVL.bP2(N);
END_STEP
TRANSITION FROM LoadTank3 TO Charge
    := GVL.fTE[14] + 3 >= GVL.fTE[17];
END_TRANSITION
TRANSITION FROM LoadTank3 TO Init
    := GVL.bValveManual;
END_TRANSITION
TRANSITION FROM Charge TO ReduceHeat
    := GVL.fTE[10] > 80 AND GVL.fTE[12] > 80 AND GVL.fTE[14] > 80;
END_TRANSITION
STEP ReduceHeat:
    GVL.bHV[9](N);
    GVL.bHV[11](N);
    GVL.bP3(N);
    GVL.bFanPower(N);
END_STEP
TRANSITION FROM ReduceHeat TO Charge
    := GVL.fTE[14] < 70;
END_TRANSITION
TRANSITION FROM ReduceHeat TO Init
    := GVL.bValveManual;
END_TRANSITION

ACTION Init_action:
(*GVL.bHV[1] := FALSE;
GVL.bHV[2] := FALSE;
GVL.bHV[3] := FALSE;
GVL.bHV[4] := FALSE;
GVL.bHV[5] := FALSE;
GVL.bHV[6] := FALSE;
GVL.bHV[7] := FALSE;
GVL.bHV[8] := FALSE;
GVL.bHV[9] := FALSE;
GVL.bHV[10] := FALSE;*)
GVL.bP2 := FALSE;
GVL.bP3 := FALSE;
END_ACTION

END_PROGRAM
